// TIA Portal V18 export
FUNCTION "FC_DI" : Void   // FC1, STL
{ S7_Optimized_Access := 'TRUE' }
VERSION : 0.1
// stored: AutoNumber true, UDAEnableTagReadback false
BEGIN

NETWORK
TITLE = 
      A     "in_SelStart";
      =     "DB_DI".in_SelStart;

      A     "in_SelStop";
      =     "DB_DI".in_SelStop;

      A     "in_BtnEmergency";
      =     "DB_DI".in_BtnEmergency;

      A     "in_BtnReset";
      =     "DB_DI".in_BtnReset;

      A     "in_Capacitive";
      =     "DB_DI".in_Capacitive;

      A     "in_5";
      =     "DB_DI".in_5;

      A     "in_6";
      =     "DB_DI".in_6;

      A     "in_PhCell_0";
      =     "DB_DI".in_PhCell_0;

      A     "in_PhCell_1";
      =     "DB_DI".in_PhCell_1;

      A     "in_PhCell_2";
      =     "DB_DI".in_PhCell_2;

      A     "in_PhCell_3";
      =     "DB_DI".in_PhCell_3;

      A     "in_PhCell_4";
      =     "DB_DI".in_PhCell_4;

      A     "in_PhCell_5";
      =     "DB_DI".in_PhCell_5;

      A     "in_PhCell_6";
      =     "DB_DI".in_PhCell_6;

      A     "in_PhCell_7";
      =     "DB_DI".in_PhCell_7;

      A     "in_PhCell_8";
      =     "DB_DI".in_PhCell_8;

      A     "in_Picker";
      =     "DB_DI".in_Picker;

      A     "in_17";
      =     "DB_DI".in_17;

      A     "in_17";
      =     "DB_DI".in_17;

      A     "in_18";
      =     "DB_DI".in_18;

      A     "in_19";
      =     "DB_DI".in_19;

      A     "in_20";
      =     "DB_DI".in_20;

      A     "in_21";
      =     "DB_DI".in_21;

      A     "in_22";
      =     "DB_DI".in_22;

      A     "in_23";
      =     "DB_DI".in_23;

      A     "in_24";
      =     "DB_DI".in_24;

      A     "in_25";
      =     "DB_DI".in_26;

      A     "in_27";
      =     "DB_DI".in_27;

      A     "in_28";
      =     "DB_DI".in_28;

      A     "in_29";
      =     "DB_DI".in_29;

      A     "in_30";
      =     "DB_DI".in_30;

      A     "in_31";
      =     "DB_DI".in_31;




//Flacos

      A     "in_BtnReset";
      FP    "Data".flanks[0];
      =     "DB_DI".BtnReset_p;

      A     "in_PhCell_0";
      FP    "Data".flanks[1];
      =     "DB_DI".PhCell_0_p;

      A     "in_PhCell_0";
      FN    "Data".flanks[2];
      =     "DB_DI".PhCell_0_n;

      A     "in_PhCell_1";
      FP    "Data".flanks[3];
      =     "DB_DI".PhCell_1_p;

      A     "in_PhCell_1";
      FN    "Data".flanks[4];
      =     "DB_DI".PhCell_1_n;

      A     "in_PhCell_2";
      FP    "Data".flanks[5];
      =     "DB_DI".PhCell_2_p;

      A     "in_PhCell_2";
      FN    "Data".flanks[6];
      =     "DB_DI".PhCell_2_n;

      A     "in_PhCell_3";
      FP    "Data".flanks[7];
      =     "DB_DI".PhCell_3_p;

      A     "in_PhCell_3";
      FN    "Data".flanks[8];
      =     "DB_DI".PhCell_3_n;

      A     "in_PhCell_4";
      FP    "Data".flanks[9];
      =     "DB_DI".PhCell_4_p;

      A     "in_PhCell_4";
      FN    "Data".flanks[10];
      =     "DB_DI".PhCell_4_n;

      A     "in_PhCell_5";
      FP    "Data".flanks[11];
      =     "DB_DI".PhCell_5_p;

      A     "in_PhCell_5";
      FN    "Data".flanks[12];
      =     "DB_DI".PhCell_5_n;

      A     "in_PhCell_6";
      FP    "Data".flanks[13];
      =     "DB_DI".PhCell_6_p;

      A     "in_PhCell_6";
      FN    "Data".flanks[14];
      =     "DB_DI".PhCell_6_n;

      A     "in_PhCell_7";
      FP    "Data".flanks[15];
      =     "DB_DI".PhCell_7_p;

      A     "in_PhCell_7";
      FN    "Data".flanks[16];
      =     "DB_DI".PhCell_7_n;

      A     "in_PhCell_8";
      FP    "Data".flanks[17];
      =     "DB_DI".PhCell_8_p;

      A     "in_PhCell_8";
      FN    "Data".flanks[18];
      =     "DB_DI".PhCell_8_n;









END_FUNCTION
